	IF NOT(bError) THEN
		ReadBlock(
			NETID 		:= sNetId,
			PORT 		:= nPort,
			IDXGRP 		:= nIDN,
			IDXOFFS 	:= iMIN,
			LEN 		:= cbRead,
			DESTADDR 	:= dwDestAddr_I,
			READ 		:= TRUE,
			TMOUT 		:= tTimeout
		);
		Timeout(IN := FALSE);
	END_IF

10:	(* read min act *)
	ReadBlock(READ := FALSE);

	IF NOT(ReadBlock.BUSY) THEN
		ReadBlock(READ := FALSE);

		IF NOT(ReadBlock.ERR) THEN
			(* done *)
			iState  := 0;
			bBusy   := FALSE;

			ReadBlock(READ := FALSE);
			iRepeats := 0;
		ELSE
			(* Timeout error *)
			IF (ReadBlock.ErrId = 16#745) AND (iRepeats <= 3) THEN
				Timeout(IN := TRUE);

				IF Timeout.Q THEN
					Timeout(IN := FALSE);
					(* retry request 3 times after timeout of 10 ms *)

					ReadBlock(READ := FALSE); (* create rising edge *)
					iRepeats := iRepeats + 1;
					iState	 := 9;
				END_IF

			(* report other errors immeditelly *)
			ELSE
				bError 	:= ReadBlock.ERR;
				nErrId  := ReadBlock.ERRID;
				bBusy   := FALSE;
				iState	:= 0;

				Timeout(IN := FALSE);
				ReadBlock(READ := FALSE);
			END_IF
		END_IF
	END_IF

11:	(* read max init *)
	iState	   	 := 12;
	dwDestAddr_I := dwDestAddr;

	CASE sAttrib.eLength OF
		eLEN_2BYTE:
			cbRead 	 := 2;

		eLEN_4BYTE:
			cbRead	 := 4;

		eLEN_8BYTE:
			cbRead	 := 8;

	ELSE
		bError	 := TRUE;
		nErrId	 := 16#1004; (* Data parameter wrong value size *)
		bBusy	 := FALSE;
		iState 	 := 0;
	END_CASE

	cbRead 	 	:= LIMIT(0, cbRead, cbLen);

	IF NOT(bError) THEN
		ReadBlock(
			NETID 		:= sNetId,
			PORT 		:= nPort,
			IDXGRP 		:= nIDN,
			IDXOFFS 	:= iMAX,
			LEN 		:= cbRead,
			DESTADDR 	:= dwDestAddr_I,
			READ 		:= TRUE,
			TMOUT 		:= tTimeout
		);
		Timeout(IN := FALSE);
	END_IF

12:	(* read max act *)
	ReadBlock(READ := FALSE);

	IF NOT(ReadBlock.BUSY) THEN
		ReadBlock(READ := FALSE);

		IF NOT(ReadBlock.ERR) THEN
			(* done *)
			iState  := 0;
			bBusy   := FALSE;

			ReadBlock(READ := FALSE);
			iRepeats := 0;
		ELSE
			(* Timeout error *)
			IF (ReadBlock.ErrId = 16#745) AND (iRepeats <= 3) THEN
				Timeout(IN := TRUE);

				IF Timeout.Q THEN
					Timeout(IN := FALSE);
					(* retry request 3 times after timeout of 10 ms *)

					ReadBlock(READ := FALSE); (* create rising edge *)
					iRepeats := iRepeats + 1;
					iState	 := 11;
				END_IF

			(* report other errors immeditelly *)
			ELSE
				bError 	:= ReadBlock.ERR;
				nErrId  := ReadBlock.ERRID;
				bBusy   := FALSE;
				iState	:= 0;

				Timeout(IN := FALSE);
				ReadBlock(READ := FALSE);
			END_IF
		END_IF
	END_IF

13: (* Function State *)
	iState 		 := 14;
	dwDestAddr_I := dwDestAddr;
	cbRead		 := cbLen;

	ReadBlock(
		NETID 		:= sNetId,
		PORT 		:= nPort,
		IDXGRP 		:= nIDN,
		IDXOFFS 	:= iFCNSTATE,
		LEN 		:= cbRead,
		DESTADDR 	:= dwDestAddr_I,
		READ 		:= TRUE,
		TMOUT 		:= tTimeout
	);
	Timeout(IN := FALSE);


14:	(* read value act *)
	ReadBlock(READ := FALSE);

	IF NOT(ReadBlock.BUSY) THEN
		ReadBlock(READ := FALSE);

		IF NOT(ReadBlock.ERR) THEN
			(* done *)
			iState	:= 0;
			bBusy	:= FALSE;
			iRepeats 	:= 0;
			ReadBlock(READ := FALSE);
		ELSE
			(* Timeout error *)
			IF (ReadBlock.ErrId = 16#745) AND (iRepeats <= 3) THEN
				Timeout(IN := TRUE);

				IF Timeout.Q THEN
					Timeout(IN := FALSE);
					(* retry request 3 times after timeout of 10 ms *)

					ReadBlock(READ := FALSE); (* create rising edge *)
					iRepeats := iRepeats + 1;
					iState	 := 13;
				END_IF

			(* report other errors immeditelly *)
			ELSE
				bError 	:= ReadBlock.ERR;
				nErrId  := ReadBlock.ERRID;
				bBusy   := FALSE;
				iState	:= 0;

				Timeout(IN := FALSE);
				ReadBlock(READ := FALSE);
			END_IF
		END_IF
	END_IF

ELSE
	(* error *)
	bError	:= TRUE;
	bBusy	:= FALSE;
	iState 	:= 0;
END_CASE

bExecute_I := bExecute;
END_FUNCTION_BLOCK

(* POU IOF_SER_IDN_Write, ST *)
FUNCTION_BLOCK IOF_SER_IDN_Write
VAR_INPUT
	sNetId 				: T_AmsNetId;
	nIDN				: UINT;					(* S: binary 0******* ********, P: binary 1******* ******** *)
	bExecute			: BOOL;					(* starts write with rising edge *)
	nPort				: UINT;					(* sercos axis ads port number *)
	nAttrib				: DWORD;				(* write: 0= Value *)
	cbLen				: UDINT;				(* max lenght of data buffer *)
	dwSrcAddr 			: DWORD;				(* address of data buffer *)
	tTimeout			: TIME := DEFAULT_ADS_TIMEOUT;(* timeout for complete parameter access (e.g. incl. attribute) *)
END_VAR
VAR_OUTPUT
	nAttribRd			: DWORD;
	sAttrib				: ST_SercosParamAttrib;
	bBusy 				: BOOL;
	bError				: BOOL;
	nErrId 				: UDINT;
END_VAR
VAR
	WriteBlock 			: ADSWRITE;
	ReadBlock 			: ADSREAD;
	iState				: INT;
	iRepeats			: INT;
	cbRead				: UDINT;
	cbWrite				: UDINT;
	dwDestAddr			: UDINT;
	nRetVal				: UDINT;
	bExecute_I			: BOOL;
	Timeout				: TON := (PT := T#100ms);
END_VAR
VAR CONSTANT
	iVALUE				: DINT := 0;		(* Parameter Value *)
	iATTRIB				: DINT := 3;		(* Parameter Attribute *)
END_VAR
(* state machine *)
CASE iState OF
0:	(* wait for rising edge *)
	IF bExecute AND NOT(bExecute_I) THEN
		bBusy    	:= TRUE;
		bError 	  	:= FALSE;
		nErrId 	  	:= 0;
		iRepeats 	:= 0;

		Timeout(IN := FALSE);
		ReadBlock(READ := FALSE);
		WriteBlock(WRITE := FALSE);

		IF (nAttrib <> 0) THEN
			sAttrib.nFactor			:= DWORD_TO_UINT(nAttrib          AND 16#0000FFFF); (* bits  0..15 *)
			sAttrib.eLength			:= DWORD_TO_INT(SHR(nAttrib,  16) AND 16#00000007);	(* bits 16..18 *)
			sAttrib.bCommand		:= DWORD_TO_BOOL(SHR(nAttrib, 19) AND 16#00000001);	(* bit  19     *)
			sAttrib.eType			:= DWORD_TO_INT(SHR(nAttrib,  20) AND 16#00000007);	(* bits 20..22 *)
			sAttrib.bReserved1		:= DWORD_TO_BOOL(SHR(nAttrib, 23) AND 16#00000001);	(* bit  23     *)
			sAttrib.nComma			:= DWORD_TO_USINT(SHR(nAttrib,24) AND 16#0000000F); (* bits 24..27 *)
			sAttrib.bWriteProtCP2	:= DWORD_TO_BOOL(SHR(nAttrib, 28) AND 16#00000001);	(* bit  28     *)
			sAttrib.bWriteProtCP3	:= DWORD_TO_BOOL(SHR(nAttrib, 29) AND 16#00000001);	(* bit  29     *)
			sAttrib.bWriteProtCP4	:= DWORD_TO_BOOL(SHR(nAttrib, 30) AND 16#00000001);	(* bit  30     *)
			sAttrib.bReserved2		:= DWORD_TO_BOOL(SHR(nAttrib, 31) AND 16#00000001);	(* bit  31     *)
		END_IF

		IF (nAttrib = 0) OR (sAttrib.eLength = 0) THEN
			(* read attrib first, write afterwards *)
			iState 		:= 1;
			nRetVal 	:= MEMSET(ADR(sAttrib), 0, SIZEOF(sAttrib));
		ELSE
			(* use known attrib, write immediatelly *)
			nAttribRd	:= nAttrib;
			iState 		:= 3;
		END_IF
	END_IF

1:	(* read attrib init *)
	iState 		:= 2;
	nAttribRd	:= 0;
	cbRead 		:= SIZEOF(nAttribRd);
	dwDestAddr 	:= ADR(nAttribRd);

	ReadBlock(
		NETID 		:= sNetId,
		PORT 		:= nPort,
		IDXGRP 		:= nIDN,
		IDXOFFS 	:= iATTRIB,
		LEN 		:= cbRead,
		DESTADDR 	:= dwDestAddr,
		READ 		:= TRUE,
		TMOUT 		:= tTimeout
	);
	Timeout(IN := FALSE);

2:	(* read attrib act *)
	ReadBlock(READ := FALSE);

	IF NOT(ReadBlock.BUSY) THEN
		ReadBlock(READ := FALSE);

		IF NOT(ReadBlock.ERR) THEN
			(* split attribute *)
			sAttrib.nFactor			:= DWORD_TO_UINT(nAttribRd          AND 16#0000FFFF); 	(* bits  0..15 *)
			sAttrib.eLength			:= DWORD_TO_INT(SHR(nAttribRd,  16) AND 16#00000007);	(* bits 16..18 *)
			sAttrib.bCommand		:= DWORD_TO_BOOL(SHR(nAttribRd, 19) AND 16#00000001);	(* bit  19     *)
			sAttrib.eType			:= DWORD_TO_INT(SHR(nAttribRd,  20) AND 16#00000007);	(* bits 20..22 *)
			sAttrib.bReserved1		:= DWORD_TO_BOOL(SHR(nAttribRd, 23) AND 16#00000001);	(* bit  23     *)
			sAttrib.nComma			:= DWORD_TO_USINT(SHR(nAttribRd,24) AND 16#0000000F);	(* bits 24..27 *)
			sAttrib.bWriteProtCP2	:= DWORD_TO_BOOL(SHR(nAttribRd, 28) AND 16#00000001);	(* bit  28     *)
			sAttrib.bWriteProtCP3	:= DWORD_TO_BOOL(SHR(nAttribRd, 29) AND 16#00000001);	(* bit  29     *)
			sAttrib.bWriteProtCP4	:= DWORD_TO_BOOL(SHR(nAttribRd, 30) AND 16#00000001);	(* bit  30     *)
			sAttrib.bReserved2		:= DWORD_TO_BOOL(SHR(nAttribRd, 31) AND 16#00000001);	(* bit  31     *)

			ReadBlock(READ := FALSE);
			iState	 := 3;
			iRepeats := 0;
		ELSE
			(* Timeout error *)
			IF (ReadBlock.ErrId = 16#745) AND (iRepeats <= 3) THEN
				Timeout(IN := TRUE);

				IF Timeout.Q THEN
					Timeout(IN := FALSE);
					(* retry request 3 times after timeout of 10 ms *)

					ReadBlock(READ := FALSE); (* create rising edge *)
					iRepeats := iRepeats + 1;
					iState 	 := 1;
				END_IF

			(* report other errors immeditelly *)
			ELSE
				bError 	:= ReadBlock.ERR;
				nErrId  := ReadBlock.ERRID;
				bBusy   := FALSE;
				iState 	:= 0;

				Timeout(IN := FALSE);
				ReadBlock( READ := FALSE );
			END_IF
		END_IF
	END_IF

3:	(* Write value init *)
	iState := 4;

	CASE sAttrib.eLength OF
		eLEN_2BYTE:
			cbWrite := 2;

		eLEN_4BYTE:
			cbWrite := 4;

		eLEN_8BYTE:
			cbWrite := 8;

		eLEN_V1BYTE, eLEN_V2BYTE, eLEN_V4BYTE, eLEN_V8BYTE:
			(* calculate number of list items *)
			cbWrite	:= 0;
			nRetVal := MEMCPY(ADR(cbWrite), dwSrcAddr, 2);
			cbWrite	:= cbWrite + 4; (* act len & max len *)

	ELSE
		bError	:= TRUE;
		nErrId	:= 16#1004; (* Data parameter wrong value size *)
		bBusy	:= FALSE;
		iState 	:= 0;
	END_CASE

	cbWrite	:= LIMIT(0, cbWrite, cbLen);

	IF NOT(bError) THEN
		WriteBlock(
			NETID 		:= sNetId,
			PORT 		:= nPort,
			IDXGRP 		:= nIDN,
			IDXOFFS 	:= iVALUE,
			LEN 		:= cbWrite,
			SRCADDR 	:= dwSrcAddr,
			WRITE 		:= TRUE,
			TMOUT 		:= tTimeout
		);
		Timeout(IN := FALSE);
	END_IF

4:	(* Write value act *)
	WriteBlock(WRITE := FALSE);

	IF NOT(WriteBlock.BUSY) THEN
		WriteBlock(WRITE := FALSE);

		IF NOT(WriteBlock.ERR) THEN
			(* done *)
			iState := 0;
			bBusy  := FALSE;

			WriteBlock(WRITE := FALSE);
			iRepeats := 0;
		ELSE
			(* Timeout error *)
			IF (WriteBlock.ErrId = 16#745) AND (iRepeats <= 3) THEN
				Timeout(IN := TRUE);

				IF Timeout.Q THEN
					Timeout(IN := FALSE);
					(* retry request 3 times after timeout of 10 ms *)

					WriteBlock(WRITE := FALSE); (* create rising edge *)
					iRepeats := iRepeats + 1;
					iState	 := 3;
				END_IF

			(* report other errors immeditelly *)
			ELSE
				bError 	:= WriteBlock.ERR;
				nErrId  := WriteBlock.ERRID;
				bBusy   := FALSE;
				iState	:= 0;

				Timeout(IN := FALSE);
				WriteBlock(WRITE := FALSE);
			END_IF
		END_IF
	END_IF

ELSE
	(* error *)
	bError	:= TRUE;
	bBusy	:= FALSE;
	iState	:= 0;
END_CASE

bExecute_I := bExecute;
END_FUNCTION_BLOCK

(* POU IOF_SER_DRIVE_BackupEx, ST *)
FUNCTION_BLOCK IOF_SER_DRIVE_BackupEx
VAR_INPUT
	bCheck				: BOOL;
	bBackup				: BOOL;
	bRestore				: BOOL;
	bCRCEnable			: BOOL;
	bStdBackupList		: BOOL 			:= TRUE;
	bUserBackupList		: BOOL;
	sNetId 					: T_AmsNetId;
	nPort					: UINT;
	sComment			: T_MaxString;
	ePath					: E_OpenPath 	:= PATH_BOOTPATH;
	sPathName			: T_MaxString 	:= 'DRIVEPAR.BIN';
	tTimeout				: TIME := DEFAULT_ADS_TIMEOUT;
	bIgnoreParamErr		: BOOL;
END_VAR
VAR_OUTPUT
	bBusy					: BOOL;
	bError					: BOOL;
	nErrId					: UDINT;
	bCheckOK				: BOOL;
	iSkippedParams			: UINT;
	iHandledParams			: UINT;
(*	Function block specific error codes:
	16#1005 = false backup parameter type 
	16#1006 = backup list was not IDN 192 (standard backup) or 0 (userdefined)
*)
END_VAR
VAR_IN_OUT
	arrList					: ST_SercosParamList;
	arrSkippedList			: ST_SercosParamErrList;
END_VAR
VAR CONSTANT
	iVALUE					: DINT := 0;
END_VAR
VAR
	ReadSercosParam			: IOF_SER_IDN_Read;
	WriteSercosParam		: IOF_SER_IDN_Write;

	OpenBackupFile			: FB_FileOpen;
	CloseBackupFile			: FB_FileClose;
	ReadBackupFile			: FB_FileRead;
	WriteBackupFile			: FB_FileWrite;

	eState					: E_SercosBackupState;

	sCheckData				: ST_SercosString;
	wCRC16_CCITT			: WORD;
	wCheckSum				: WORD;

	bCheck_I				: BOOL;
	bBackup_I				: BOOL;
	bRestore_I				: BOOL;
	bCheck_L				: BOOL;
	bBackup_L				: BOOL;
	bRestore_L				: BOOL;
	bUpdateCRC				: BOOL;

	bBackupDone				: BOOL;
	bRestoreDone			: BOOL;

	nListArrIdx				: UINT;
	sListAttrib				: ST_SercosParamAttrib;

	cbLen					: UDINT;
	arrData					: ARRAY [0..65535] OF BYTE;

	nIDN					: UINT;
	nCRCIDN					: UINT := 142;
	bCRCIDNExist			: BOOL;
	bCRCIDNTest				: BOOL := TRUE;
	iIdx					: UINT;

	sParamHeader			: ST_SercosParamHeader;
	cbSize					: UDINT;
	sFileHeader				: ST_SercosFileHeader;
	sParamData				: ST_SercosParamData;

	iActListItem			: UINT;
	iLastListItem			: UINT;
	bEndOfList				: BOOL;

	bFileOpen				: BOOL;
	hFile					: UINT;
	nVersion				: UDINT := 1;
	nRetVal					: UDINT;

	bWrongListType			: BOOL;
	bFileError				: BOOL;
	nFileErrId				: UDINT;
	bIdnError				: BOOL;
	nIdnErrId				: UDINT;
	nIdnAccessId			: UINT;
	iLargeParam				: UINT;
END_VAR
VAR PERSISTENT
	wSavedCRC16_CCITT		: WORD;
	wSavedCheckSum			: WORD;
	sSavedCheckData			: ST_SercosString;
END_VAR
(* state machine *)
CASE eState OF
	eBkup_IDLE:
		bBusy 		 		:= FALSE;

		(* wait for command *)
		IF bCheck AND bCRCIDNTest AND bCRCEnable THEN
			bError			:= FALSE;
			nErrId			:= 0;
			bFileOpen		:= FALSE;
			bFileError		:= FALSE;
			nFileErrId		:= 0;
			bWrongListType	:= FALSE;
			bIdnError		:= FALSE;
			nIdnErrId		:= 0;
			nIdnAccessId	:= 0;
			bEndOfList		:= FALSE;
			eState 			:= eBkup_READ_IDNLIST_INI;
			bBusy			:= TRUE;
			bCheckOK 		:= FALSE;
			iSkippedParams	:= 0;
			iHandledParams	:= 0;
			iLargeParam		:= 0;
			bBackupDone		:= FALSE;
			bRestoreDone	:= FALSE;
			MEMSET(ADR(arrSkippedList), 0, SIZEOF(arrSkippedList));

		ELSIF (bCheck AND NOT(bCheck_I)) AND bCRCEnable AND bCRCIDNExist THEN
			bError			:= FALSE;
			nErrId			:= 0;
			bFileOpen		:= FALSE;
			bFileError		:= FALSE;
			nFileErrId		:= 0;
			bWrongListType	:= FALSE;
			bIdnError		:= FALSE;
			nIdnErrId		:= 0;
			nIdnAccessId	:= 0;
			bEndOfList		:= FALSE;
			eState 			:= eBkup_CHECK_CRC_ACT;
			bBusy			:= TRUE;
			bCheckOK 		:= FALSE;
			bCheck_I 		:= TRUE;
			iSkippedParams	:= 0;
			iHandledParams	:= 0;
			iLargeParam		:= 0;
			bBackupDone		:= FALSE;
			bRestoreDone	:= FALSE;
			MEMSET(ADR(arrSkippedList), 0, SIZEOF(arrSkippedList));

			ReadSercosParam(bExecute := FALSE);
			ReadSercosParam(
				sNetId 		:= sNetId,
				nIDN		:= nCRCIDN,
				bExecute	:= TRUE,
				nMode		:= iVALUE,
				nPort		:= nPort,
				nAttrib		:= 0,
				cbLen		:= SIZEOF(sCheckData),
				dwDestAddr 	:= ADR(sCheckData),
				tTimeout	:= tTimeout
			);
		ELSE
			IF (bBackup AND NOT(bBackup_I)) OR (bRestore AND NOT(bRestore_I)) THEN
				bBackup_L		:= FALSE;
				bRestore_L		:= FALSE;
				bBusy			:= FALSE;
				bError			:= FALSE;
				nErrId			:= 0;
				bFileOpen		:= FALSE;
				bFileError		:= FALSE;
				nFileErrId		:= 0;
				bWrongListType	:= FALSE;
				bIdnError		:= FALSE;
				nIdnErrId		:= 0;
				nIdnAccessId	:= 0;
				bEndOfList		:= FALSE;
				eState 			:= eBkup_READ_IDNLIST_INI;
				bBusy			:= TRUE;
				bUpdateCRC		:= TRUE;
				bCheckOK 		:= FALSE;
				iSkippedParams	:= 0;
				iHandledParams	:= 0;
				iLargeParam		:= 0;
				bBackupDone		:= FALSE;
				bRestoreDone	:= FALSE;
				MEMSET(ADR(arrSkippedList), 0, SIZEOF(arrSkippedList));

				(* initialize CRC16-CCITT and CheckSum *)
				wSavedCRC16_CCITT 			:= 16#FFFF;
				wSavedCheckSum	  			:= 16#0000;
				sSavedCheckData.iActSize	:= 0;
				sSavedCheckData.sString		:= '';

				IF bBackup AND NOT(bBackup_I) THEN
					(* latch backup request *)
					bBackup_L	:= TRUE;
					bRestore_L	:= FALSE;
					bBackup_I 	:= TRUE;

					IF bUserBackupList THEN
						(* calculate number of list items *)
						iLastListItem 	:= arrList.iActCount;
						iLastListItem 	:= iLastListItem / 2;
						iLastListItem 	:= LIMIT(0, iLastListItem, 2047);
						iActListItem	:= 0;
						nListArrIdx		:= 0;
						eState 			:= eBkup_FILEOPEN;

						OpenBackupFile(
							sNetId 		:= sNetId,
							sPathName	:= sPathName,
							nMode		:= FOPEN_MODEWRITE OR FOPEN_MODEBINARY,
							ePath		:= ePath,
							bExecute	:= TRUE,
							tTimeout	:= tTimeout
						);
					END_IF

				ELSIF bRestore AND NOT(bRestore_I) THEN
					(* latch restore request *)
					bBackup_L	:= FALSE;
					bRestore_L	:= TRUE;
					bRestore_I	:= TRUE;

					IF bUserBackupList THEN
						(* calculate number of list items *)
						iLastListItem 	:= arrList.iActCount;
						iLastListItem 	:= iLastListItem / 2;
						iLastListItem 	:= LIMIT(0, iLastListItem, 2047);
						iActListItem	:= 0;
						nListArrIdx		:= 0;
						eState 			:= eBkup_FILEOPEN;

						OpenBackupFile(
							sNetId 		:= sNetId,
							sPathName	:= sPathName,
							nMode		:= FOPEN_MODEREAD OR FOPEN_MODEBINARY,
							ePath		:= ePath,
							bExecute	:= TRUE,
							tTimeout	:= tTimeout
						);
					END_IF
				END_IF
			END_IF
		END_IF

		wCRC16_CCITT 		:= wSavedCRC16_CCITT;
		wCheckSum	 		:= wSavedCheckSum;


	(*** check CRC and CheckSum ***)
	eBkup_CHECK_CRC_ACT:
		ReadSercosParam(bExecute := FALSE);

		IF NOT(ReadSercosParam.bBusy) THEN
			(* not busy anymore *)
			bError	:= ReadSercosParam.bError;
			nErrId	:= ReadSercosParam.nErrId;
			ReadSercosParam(bExecute := FALSE);

			IF bError THEN
				(* error *)
				bIdnError		:= TRUE;
				nIdnErrId		:= nErrId;
				nIdnAccessId	:= nCRCIDN;
				bBusy			:= FALSE;
				eState 			:= eBkup_IDLE;
			ELSE
				(* read done, compare string *)
				bCheckOK 		:= (sCheckData.sString = sSavedCheckData.sString) AND (sCheckData.sString <> '');
				bBusy			:= FALSE;
				eState 			:= eBkup_IDLE;
			END_IF
		END_IF


	(*** read parameter list ***)
	eBkup_READ_IDNLIST_INI:
		(* first scan: initialization with rising edge on bExecute *)
		eState 			:= eBkup_READ_IDNLIST_ACT;

		IF bStdBackupList AND NOT(bCRCIDNTest) THEN
			nIDN		:= 192;
		ELSE
			nIDN		:= 17;
		END_IF

		ReadSercosParam(bExecute := FALSE);
		ReadSercosParam(
			sNetId 		:= sNetId,
			nIDN		:= nIDN,
			bExecute	:= TRUE,
			nMode		:= iVALUE,
			nPort		:= nPort,
			nAttrib		:= 0,
			cbLen		:= SIZEOF(arrList),
			dwDestAddr 	:= ADR(arrList),
			tTimeout	:= tTimeout
		);

	eBkup_READ_IDNLIST_ACT:
		(* following scans: wait for not busy *)
		ReadSercosParam(bExecute := FALSE);

		IF NOT(ReadSercosParam.bBusy) THEN
			(* not busy anymore *)
			bError	:= ReadSercosParam.bError;
			nErrId	:= ReadSercosParam.nErrId;
			ReadSercosParam(bExecute := FALSE);

			IF bError THEN
				(* error *)
				bBackupDone		:= FALSE;
				bRestoreDone	:= FALSE;
				bBackup_L	 	:= FALSE;
				bRestore_L	 	:= FALSE;
				bBusy			:= FALSE;
				eState 			:= eBkup_IDLE;
				bIdnError		:= TRUE;
				nIdnErrId		:= nErrId;
				nIdnAccessId	:= nIDN;
			ELSE
				(* done *)
				sListAttrib		:= ReadSercosParam.sAttrib;

				IF (sListAttrib.eType = eType_ID) AND (sListAttrib.eLength = eLEN_V2BYTE) THEN
					(* calculate number of list items *)
					iLastListItem 	:= arrList.iActCount;
					iLastListItem 	:= iLastListItem / 2;
					iLastListItem 	:= LIMIT(0, iLastListItem, 2047);
					iActListItem	:= 0;
					nListArrIdx		:= 0;

					IF bCRCIDNTest THEN
						bCRCIDNTest  := FALSE;
						bCRCIDNExist := FALSE;

						FOR iIdx := 0 TO iLastListItem DO
							iActListItem := arrList.iList[iIdx];

							IF iActListItem = nCRCIDN THEN
								bCRCIDNExist := TRUE;
								EXIT;
							END_IF
						END_FOR

						IF bBackup_L OR bRestore_L THEN
							eState 	:= eBkup_READ_IDNLIST_INI;
						ELSE
							bBusy	:= FALSE;
							eState 	:= eBkup_IDLE;
						END_IF

					ELSE
						IF bBackup_L THEN
							eState 		:= eBkup_FILEOPEN;

							OpenBackupFile(
								sNetId 		:= sNetId,
								sPathName	:= sPathName,
								nMode		:= FOPEN_MODEWRITE OR FOPEN_MODEBINARY,
								ePath		:= ePath,
								bExecute	:= TRUE,
								tTimeout	:= tTimeout
							);

						ELSIF bRestore_L THEN
							eState 		:= eBkup_FILEOPEN;

							OpenBackupFile(
								sNetId 		:= sNetId,
								sPathName	:= sPathName,
								nMode		:= FOPEN_MODEREAD OR FOPEN_MODEBINARY,
								ePath		:= ePath,
								bExecute	:= TRUE,
								tTimeout	:= tTimeout
							);
						ELSE
							bBusy			:= FALSE;
							eState 			:= eBkup_IDLE;
						END_IF
					END_IF
				ELSE
					bBackupDone		:= FALSE;
					bRestoreDone	:= FALSE;
					bBackup_L	 	:= FALSE;
					bRestore_L	 	:= FALSE;
					bError			:= TRUE;
					nErrId			:= 16#1005;
					bBusy			:= FALSE;
					eState 			:= eBkup_IDLE;
				END_IF
			END_IF
		END_IF


	(*** backup current list ***)
	eBkup_FILEOPEN:
		OpenBackupFile(bExecute	:= FALSE);

		IF NOT(OpenBackupFile.bBusy) THEN
			bError	:= OpenBackupFile.bError;
			nErrId	:= OpenBackupFile.nErrId;
			OpenBackupFile(bExecute	:= FALSE);

			IF bError THEN
				(* error *)
				bBackupDone	:= FALSE;
				bRestoreDone:= FALSE;
				bBackup_L	:= FALSE;
				bRestore_L	:= FALSE;
				nFileErrId	:= nErrId;
				bBusy		:= FALSE;
				eState 		:= eBkup_IDLE;
				bFileOpen	:= FALSE;
				hFile		:= 0;
			ELSE
				bFileOpen	:= TRUE;
				hFile		:= OpenBackupFile.hFile;

				IF bBackup_L THEN
					(* preset header *)
					sFileHeader.nVersion 	 := nVersion;
					IF bUserBackupList THEN
						sFileHeader.nListType 	 := 0;
					ELSE
						sFileHeader.nListType 	 := nIDN;
					END_IF
					sFileHeader.cbCommentLen := SIZEOF(sComment);
					nRetVal 				 := MEMCPY(ADR(sFileHeader.sComment), ADR(sComment), SIZEOF(sComment));

					WriteBackupFile(
						sNetId 		:= sNetId,
						hFile		:= hFile,
						pWriteBuff	:= ADR(sFileHeader),
						cbWriteLen	:= SIZEOF(sFileHeader),
						bExecute	:= TRUE,
						tTimeout	:= tTimeout
					);
					eState 	:= eBkup_BACKUP_WRITE_FILEHEADER;

				ELSIF bRestore_L THEN
					nRetVal := MEMSET(ADR(sFileHeader), 0, SIZEOF(sFileHeader));

					(* load header *)
					ReadBackupFile(
						sNetId 		:= sNetId,
						hFile		:= hFile,
						pReadBuff	:= ADR(sFileHeader),
						cbReadLen	:= SIZEOF(sFileHeader),
						bExecute	:= TRUE,
						tTimeout	:= tTimeout
					);
					eState 	:= eBkup_RESTORE_READ_FILEHEADER;
				END_IF
			END_IF
		END_IF


	(*** backup init ***)
	eBkup_BACKUP_WRITE_FILEHEADER:
		WriteBackupFile(bExecute := FALSE);

		IF NOT(WriteBackupFile.bBusy) THEN
			bError	:= WriteBackupFile.bError;
			nErrId	:= WriteBackupFile.nErrId;
			WriteBackupFile(bExecute := FALSE);

			IF bError THEN
				(* error *)
				bBackupDone	:= FALSE;
				bFileError	:= TRUE;
				nFileErrId	:= nErrId;
				bError		:= FALSE;
				nErrId		:= 0;
				eState 		:= eBkup_FILECLOSE;

				(* backup aborted *)
				CloseBackupFile(
					sNetId 		:= sNetId,
					hFile		:= hFile,
					bExecute	:= TRUE,
					tTimeout	:= tTimeout
				);

			ELSE
				cbSize 	:= WriteBackupFile.cbWrite;
				eState 	:= eBkup_BACKUP_PARAM_INI;
			END_IF
		END_IF

	(* backup current list *)
	eBkup_BACKUP_PARAM_INI:
		IF NOT(bEndOfList) THEN
			(* first scan: initialization with rising edge on bBackup *)
			bBackupDone			:= FALSE;

			(* get parameter *)
			IF (nListArrIdx >= 0) AND (nListArrIdx <= 2047) THEN
				eState 			:= eBkup_BACKUP_PARAM_ACT;
				nIDN 			:= arrList.iList[nListArrIdx];
				nListArrIdx		:= nListArrIdx + 1;

				ReadSercosParam(bExecute := FALSE);
				ReadSercosParam(
					sNetId 		:= sNetId,
					nIDN		:= nIDN,
					bExecute	:= TRUE,
					nMode		:= iVALUE,
					nPort		:= nPort,
					nAttrib		:= 0,
					cbLen		:= SIZEOF(arrData),
					dwDestAddr 	:= ADR(arrData),
					tTimeout	:= tTimeout
				);

			ELSE
				(* wrong index *)
				ReadSercosParam(bExecute := FALSE);
				iActListItem	:= 0;
				bBackupDone		:= FALSE;
				bIdnError		:= TRUE;
				bError			:= FALSE;
				nErrId			:= 0;
				eState 			:= eBkup_FILECLOSE;

				(* backup aborted *)
				CloseBackupFile(
					sNetId 		:= sNetId,
					hFile		:= hFile,
					bExecute	:= TRUE,
					tTimeout	:= tTimeout
				);
			END_IF
		ELSE
			(* backup completed *)
			ReadSercosParam(bExecute := FALSE);
			iActListItem	:= 0;
			eState 			:= eBkup_FILECLOSE;

			CloseBackupFile(
				sNetId 		:= sNetId,
				hFile		:= hFile,
				bExecute	:= TRUE,
				tTimeout	:= tTimeout
			);
		END_IF

	eBkup_BACKUP_PARAM_ACT:
		(* following scans: wait for not busy *)
		ReadSercosParam(bExecute := FALSE);

		IF NOT(ReadSercosParam.bBusy) THEN
			(* not busy anymore *)
			bError				:= ReadSercosParam.bError;
			nErrId				:= ReadSercosParam.nErrId;
			ReadSercosParam(bExecute := FALSE);

			IF bError AND NOT bIgnoreParamErr THEN
				(* error *)
				bBackupDone		:= FALSE;
				bRestoreDone	:= FALSE;
				bIdnError		:= TRUE;
				nIdnErrId		:= nErrId;
				nIdnAccessId	:= nIDN;
				bError			:= FALSE;
				nErrId			:= 0;
				eState 			:= eBkup_FILECLOSE;

				(* backup aborted *)
				CloseBackupFile(
					sNetId 		:= sNetId,
					hFile		:= hFile,
					bExecute	:= TRUE,
					tTimeout	:= tTimeout
				);
			ELSE
				IF NOT bError THEN
					(* save data header *)
					sParamHeader.nIDN	:= ReadSercosParam.nIDN;
					sParamHeader.nAttrib:= ReadSercosParam.nAttribRd;
					sParamHeader.cbSize	:= UDINT_TO_UINT(ReadSercosParam.cbRead);

					IF sParamHeader.cbSize > 4095 THEN
						iLargeParam := iLargeParam + 1;
					END_IF

					(* update CRC16-CCITT and CheckSum *)
					IF nIDN <> nCRCIDN THEN
						wCRC16_CCITT	:= F_CRC16_CCITT(ADR(arrData), sParamHeader.cbSize, wCRC16_CCITT);
						wCheckSum		:= F_CheckSum16(ADR(arrData), sParamHeader.cbSize, wCheckSum);
					END_IF

					WriteBackupFile(
						sNetId 		:= sNetId,
						hFile		:= hFile,
						pWriteBuff	:= ADR(sParamHeader),
						cbWriteLen	:= SIZEOF(sParamHeader),
						bExecute	:= TRUE,
						tTimeout	:= tTimeout
					);

					eState 		:= eBkup_BACKUP_WRITE_HEADER;
				ELSE
					(* ignore param read error *)
					IF iSkippedParams < 2047 THEN
						arrSkippedList.iList[iSkippedParams] := nIDN;
						arrSkippedList.iError[iSkippedParams] := ReadSercosParam.nErrId;
						arrSkippedList.iActCount := arrSkippedList.iActCount + 1;
						arrSkippedList.iMaxCount := arrSkippedList.iActCount;
					END_IF
					iSkippedParams := iSkippedParams + 1;

					(* next item *)
					IF NOT(bEndOfList) THEN
						(* next item *)
						iActListItem		:= iActListItem + 1;
	
						(* backup next parameter *)
						eState 				:= eBkup_BACKUP_PARAM_INI;
	
						IF (iActListItem >= iLastListItem) THEN
							iActListItem	:= 0;
							bEndOfList		:= TRUE;
	
							(* backup completed *)
							ReadSercosParam(bExecute := FALSE);
							CloseBackupFile(
								sNetId 		:= sNetId,
								hFile		:= hFile,
								bExecute	:= TRUE,
								tTimeout	:= tTimeout
							);
							eState 		:= eBkup_FILECLOSE;
						END_IF
					ELSE
						(* backup completed *)
						CloseBackupFile(
							sNetId 		:= sNetId,
							hFile		:= hFile,
							bExecute	:= TRUE,
							tTimeout	:= tTimeout
						);
						ReadSercosParam(bExecute := FALSE);
						eState 		:= eBkup_FILECLOSE;
					END_IF
				END_IF
			END_IF
		END_IF

	eBkup_BACKUP_WRITE_HEADER:
		WriteBackupFile(bExecute := FALSE);

		IF NOT(WriteBackupFile.bBusy) THEN
			bError	:= WriteBackupFile.bError;
			nErrId	:= WriteBackupFile.nErrId;
			WriteBackupFile(bExecute := FALSE);

			IF bError THEN
				(* error *)
				bBackupDone	:= FALSE;
				bFileError	:= TRUE;
				nFileErrId	:= nErrId;
				bError		:= FALSE;
				nErrId		:= 0;
				eState 		:= eBkup_FILECLOSE;

				(* backup aborted *)
				CloseBackupFile(
					sNetId 		:= sNetId,
					hFile		:= hFile,
					bExecute	:= TRUE,
					tTimeout	:= tTimeout
				);
			ELSE
				cbSize := WriteBackupFile.cbWrite;

				(* save data *)
				CASE sParamData.sAttrib.eLength OF
					eLEN_2BYTE,  eLEN_4BYTE,  eLEN_8BYTE,
					eLEN_V1BYTE, eLEN_V2BYTE, eLEN_V4BYTE, eLEN_V8BYTE:
						WriteBackupFile(
							sNetId 		:= sNetId,
							hFile		:= hFile,
							pWriteBuff	:= ADR(arrData),
							cbWriteLen	:= sParamHeader.cbSize,
							bExecute	:= TRUE,
							tTimeout	:= tTimeout
						);
				ELSE
					;
				END_CASE

				eState 		:= eBkup_BACKUP_WRITE_DATA;
			END_IF
		END_IF

	eBkup_BACKUP_WRITE_DATA:
		WriteBackupFile(bExecute := FALSE);

		IF NOT(WriteBackupFile.bBusy) THEN
			bError	:= WriteBackupFile.bError;
			nErrId	:= WriteBackupFile.nErrId;
			WriteBackupFile(bExecute := FALSE);

			IF bError THEN
				(* error *)
				bBackupDone	:= FALSE;
				bFileError	:= TRUE;
				nFileErrId	:= nErrId;
				bError		:= FALSE;
				nErrId		:= 0;
				eState 		:= eBkup_FILECLOSE;

				(* backup aborted *)
				CloseBackupFile(
					sNetId 		:= sNetId,
					hFile		:= hFile,
					bExecute	:= TRUE,
					tTimeout	:= tTimeout
				);
			ELSE
				cbSize 		:= WriteBackupFile.cbWrite;
				iHandledParams	:= iHandledParams + 1;

				(* next item *)
				IF NOT(bEndOfList) THEN
					(* next item *)
					iActListItem		:= iActListItem + 1;

					(* backup next parameter *)
					eState 				:= eBkup_BACKUP_PARAM_INI;

					IF (iActListItem >= iLastListItem) THEN
						iActListItem	:= 0;
						bEndOfList		:= TRUE;

						(* backup completed *)
						ReadSercosParam(bExecute := FALSE);
						CloseBackupFile(
							sNetId 		:= sNetId,
							hFile		:= hFile,
							bExecute	:= TRUE,
							tTimeout	:= tTimeout
						);
						eState 		:= eBkup_FILECLOSE;
					END_IF
				ELSE
					(* backup completed *)
					CloseBackupFile(
						sNetId 		:= sNetId,
						hFile		:= hFile,
						bExecute	:= TRUE,
						tTimeout	:= tTimeout
					);
					ReadSercosParam(bExecute := FALSE);
					eState 		:= eBkup_FILECLOSE;
				END_IF
			END_IF
		END_IF


	(*** restore init ***)
	eBkup_RESTORE_READ_FILEHEADER:
		ReadBackupFile(bExecute := FALSE);

		IF NOT(ReadBackupFile.bBusy) THEN
			bError	:= ReadBackupFile.bError;
			nErrId	:= ReadBackupFile.nErrId;
			ReadBackupFile(bExecute := FALSE);

			IF bError THEN
				(* error *)
				bRestoreDone:= FALSE;
				bFileError	:= TRUE;
				nFileErrId	:= nErrId;
				bError		:= FALSE;
				nErrId		:= 0;
				eState 		:= eBkup_FILECLOSE;

				(* backup aborted *)
				CloseBackupFile(
					sNetId 		:= sNetId,
					hFile		:= hFile,
					bExecute	:= TRUE,
					tTimeout	:= tTimeout
				);
			ELSE
				cbSize 			:= ReadBackupFile.cbRead;
				sComment		:= sFileHeader.sComment;

				IF sFileHeader.nListType = 192 OR sFileHeader.nListType = 0 THEN
					bWrongListType	:= FALSE;

					ReadBackupFile(
						sNetId 		:= sNetId,
						hFile		:= hFile,
						pReadBuff	:= ADR(sParamHeader),
						cbReadLen	:= SIZEOF(sParamHeader),
						bExecute	:= TRUE,
						tTimeout	:= tTimeout
					);
					eState 			:= eBkup_RESTORE_READ_HEADER;
				ELSE
					bWrongListType	:= TRUE;

					(* backup completed *)
					CloseBackupFile(
						sNetId 		:= sNetId,
						hFile		:= hFile,
						bExecute	:= TRUE,
						tTimeout	:= tTimeout
					);
					eState 		:= eBkup_FILECLOSE;
				END_IF
			END_IF
		END_IF

	eBkup_RESTORE_READ_HEADER:
		ReadBackupFile(bExecute := FALSE);

		IF NOT(ReadBackupFile.bBusy) THEN
			bError	:= ReadBackupFile.bError;
			nErrId	:= ReadBackupFile.nErrId;
			ReadBackupFile(bExecute := FALSE);

			IF bError THEN
				(* error *)
				bRestoreDone:= FALSE;
				bFileError	:= TRUE;
				nFileErrId	:= nErrId;
				bError		:= FALSE;
				nErrId		:= 0;
				eState 		:= eBkup_FILECLOSE;

				(* backup aborted *)
				CloseBackupFile(
					sNetId 		:= sNetId,
					hFile		:= hFile,
					bExecute	:= TRUE,
					tTimeout	:= tTimeout
				);
			ELSE
				cbSize := sParamHeader.cbSize;

				IF (ReadBackupFile.cbRead <> 0) THEN
					nRetVal		:= MEMSET(ADR(arrData[0]), 0, SIZEOF(arrData));

					ReadBackupFile(
						sNetId 		:= sNetId,
						hFile		:= hFile,
						pReadBuff	:= ADR(arrData),
						cbReadLen	:= sParamHeader.cbSize,
						bExecute	:= TRUE,
						tTimeout	:= tTimeout
					);
					eState 			:= eBkup_RESTORE_READ_DATA;
				ELSE
					(* backup completed *)
					CloseBackupFile(
						sNetId 		:= sNetId,
						hFile		:= hFile,
						bExecute	:= TRUE,
						tTimeout	:= tTimeout
					);
					bEndOfList	:= TRUE;
					eState 		:= eBkup_FILECLOSE;
				END_IF
			END_IF
		END_IF

	eBkup_RESTORE_READ_DATA:
		ReadBackupFile(bExecute := FALSE);

		IF NOT(ReadBackupFile.bBusy) THEN
			bError		:= ReadBackupFile.bError;
			nErrId		:= ReadBackupFile.nErrId;
			ReadBackupFile(bExecute := FALSE);

			IF bError THEN
				(* error *)
				bRestoreDone:= FALSE;
				bFileError	:= TRUE;
				nFileErrId	:= nErrId;
				bError		:= FALSE;
				nErrId		:= 0;
				eState 		:= eBkup_FILECLOSE;

				(* backup aborted *)
				CloseBackupFile(
					sNetId 		:= sNetId,
					hFile		:= hFile,
					bExecute	:= TRUE,
					tTimeout	:= tTimeout
				);
			ELSE
				IF ReadBackupFile.bEOF THEN
					bEndOfList	:= TRUE;
				END_IF

				cbSize 	:= ReadBackupFile.cbRead;
				eState 	:= eBkup_RESTORE_PARAM_INI;
			END_IF
		END_IF

	(* restore current list item *)
	eBkup_RESTORE_PARAM_INI:
		(* first scan: initialization with rising edge on bBackup *)
		bRestoreDone	:= FALSE;
		eState 			:= eBkup_RESTORE_PARAM_ACT;
		nIDN			:= sParamHeader.nIDN;

		sParamData.nAttrib					:= sParamHeader.nAttrib;

		(* split attribute *)
		sParamData.sAttrib.nFactor			:= DWORD_TO_UINT(sParamHeader.nAttrib AND 16#0000FFFF); 			(* bits  0..15 *)
		sParamData.sAttrib.eLength			:= DWORD_TO_INT(SHR(sParamHeader.nAttrib, 16) AND 16#00000007);		(* bits 16..18 *)
		sParamData.sAttrib.bCommand			:= DWORD_TO_BOOL(SHR(sParamHeader.nAttrib, 19) AND 16#00000001);	(* bit  19     *)
		sParamData.sAttrib.eType			:= DWORD_TO_INT(SHR(sParamHeader.nAttrib, 20) AND 16#00000007);		(* bits 20..22 *)
		sParamData.sAttrib.bReserved1		:= DWORD_TO_BOOL(SHR(sParamHeader.nAttrib, 23) AND 16#00000001);	(* bit  23     *)
		sParamData.sAttrib.nComma			:= DWORD_TO_USINT(SHR(sParamHeader.nAttrib, 24) AND 16#0000000F);	(* bits 24..27 *)
		sParamData.sAttrib.bWriteProtCP2	:= DWORD_TO_BOOL(SHR(sParamHeader.nAttrib, 28) AND 16#00000001);	(* bit  28     *)
		sParamData.sAttrib.bWriteProtCP3	:= DWORD_TO_BOOL(SHR(sParamHeader.nAttrib, 29) AND 16#00000001);	(* bit  29     *)
		sParamData.sAttrib.bWriteProtCP4	:= DWORD_TO_BOOL(SHR(sParamHeader.nAttrib, 30) AND 16#00000001);	(* bit  30     *)
		sParamData.sAttrib.bReserved2		:= DWORD_TO_BOOL(SHR(sParamHeader.nAttrib, 31) AND 16#00000001);	(* bit  31     *)

		CASE sParamData.sAttrib.eLength OF
			eLEN_2BYTE:
				cbLen	:= 2;

			eLEN_4BYTE:
				cbLen	:= 4;

			eLEN_8BYTE:
				cbLen	:= 8;

			eLEN_V1BYTE, eLEN_V2BYTE, eLEN_V4BYTE, eLEN_V8BYTE:
				nRetVal := MEMCPY(ADR(cbLen), ADR(arrData), 2);
				cbLen	:= cbLen + 4; (* act len & max len *)
		ELSE
			cbLen	:= 0;
		END_CASE

		WriteSercosParam(bExecute := FALSE);
		WriteSercosParam(
			sNetId 		:= sNetId,
			nIDN		:= nIDN,
			bExecute	:= TRUE,
			nPort		:= nPort,
			nAttrib		:= sParamData.nAttrib,
			cbLen		:= cbLen,
			dwSrcAddr	:= ADR(arrData),
			tTimeout	:= tTimeout
		);

	eBkup_RESTORE_PARAM_ACT:
		(* following scans: wait for not busy *)
		WriteSercosParam(bExecute := TRUE);

		IF NOT(WriteSercosParam.bBusy) THEN
			(* not busy anymore *)
			bError				:= WriteSercosParam.bError;
			nErrId				:= WriteSercosParam.nErrId;
			WriteSercosParam(bExecute := FALSE);

			IF bError AND NOT bIgnoreParamErr THEN
				(* error *)
				bBackupDone		:= FALSE;
				bRestoreDone	:= FALSE;
				bIdnError		:= TRUE;
				nIdnErrId		:= nErrId;
				nIdnAccessId	:= nIDN;
				bError			:= FALSE;
				nErrId			:= 0;
				eState 			:= eBkup_FILECLOSE;

				(* backup aborted *)
				CloseBackupFile(
					sNetId 		:= sNetId,
					hFile		:= hFile,
					bExecute	:= TRUE,
					tTimeout	:= tTimeout
				);

			ELSE
				IF NOT bError THEN
					iHandledParams	:= iHandledParams + 1;

					IF cbLen > 4095 THEN
						iLargeParam := iLargeParam + 1;
					END_IF

					(* update CRC16-CCITT and CheckSum *)
					IF nIDN <> nCRCIDN THEN
						wCRC16_CCITT	:= F_CRC16_CCITT(ADR(arrData), cbLen, wCRC16_CCITT);
						wCheckSum		:= F_CheckSum16(ADR(arrData), cbLen, wCheckSum);
					END_IF
				ELSE
					(* ignore param write error *)
					IF iSkippedParams < 2047 THEN
						arrSkippedList.iList[iSkippedParams] := nIDN;
						arrSkippedList.iError[iSkippedParams] := WriteSercosParam.nErrId;
						arrSkippedList.iActCount := arrSkippedList.iActCount + 1;
						arrSkippedList.iMaxCount := arrSkippedList.iActCount;
					END_IF
					iSkippedParams := iSkippedParams + 1;
				END_IF

				(* next parameter *)
				iActListItem	:= iActListItem + 1;

				IF NOT(bEndOfList) THEN
					ReadBackupFile(
						sNetId 		:= sNetId,
						hFile		:= hFile,
						pReadBuff	:= ADR(sParamHeader),
						cbReadLen	:= SIZEOF(sParamHeader),
						bExecute	:= TRUE,
						tTimeout	:= tTimeout
					);
					eState 			:= eBkup_RESTORE_READ_HEADER;
				ELSE
					(* backup completed *)
					CloseBackupFile(
						sNetId 		:= sNetId,
						hFile		:= hFile,
						bExecute	:= TRUE,
						tTimeout	:= tTimeout
					);
					WriteSercosParam(bExecute := FALSE);
					eState 		:= eBkup_FILECLOSE;
				END_IF
			END_IF
		END_IF

	(*** done or aborted  ***)
	eBkup_FILECLOSE:
		CloseBackupFile(bExecute := FALSE);

		IF NOT(CloseBackupFile.bBusy) THEN
			bError	:= CloseBackupFile.bError;
			nErrId	:= CloseBackupFile.nErrId;
			CloseBackupFile(bExecute := FALSE);

			IF bError THEN
				(* error *)
				bBackupDone	:= FALSE;
				bRestoreDone:= FALSE;
				bBackup_L	:= FALSE;
				bRestore_L	:= FALSE;
				bBusy		:= FALSE;
				eState 		:= eBkup_IDLE;
			ELSE
				bFileOpen	:= FALSE;
				hFile		:= 0;

				IF bUpdateCRC AND bCRCEnable THEN
					IF NOT(bFileError OR bIdnError) THEN
						sCheckData.sString := 'CRC= ';
						sCheckData.sString := CONCAT(sCheckData.sString, WORD_TO_STRING(wCRC16_CCITT));
						sCheckData.sString := CONCAT(sCheckData.sString, ', ChkSum= ');
						sCheckData.sString := CONCAT(sCheckData.sString, WORD_TO_STRING(wCheckSum));

						IF bBackup_L OR (bRestore_L AND NOT(bWrongListType)) THEN
							ReadSercosParam(bExecute := FALSE);
							ReadSercosParam(
								sNetId 		:= sNetId,
								nIDN		:= nCRCIDN,
								bExecute	:= TRUE,
								nMode		:= iVALUE,
								nPort		:= nPort,
								nAttrib		:= 0,
								cbLen		:= 4,
								dwDestAddr 	:= ADR(sCheckData),
								tTimeout	:= tTimeout
							);

							eState		 := eBkup_UPDT_CRC_INI;
						ELSE
							IF bWrongListType THEN
								bBackupDone := FALSE;
								bRestoreDone:= FALSE;
								bBackup_L	:= FALSE;
								bRestore_L	:= FALSE;
								bError		:= TRUE;
								nErrId		:= 16#1006;	(* backup list was NOT IDN 192 *)
								bBusy		:= FALSE;
								eState 		:= eBkup_IDLE;
							END_IF
						END_IF
					END_IF
				ELSE
					(* done, no CRC and check sum *)
					IF bBackup_L THEN
						bBackup_L	:= FALSE;
						bBackupDone	:= TRUE;
					ELSIF bRestore_L THEN
						bRestore_L	:= FALSE;
						IF NOT bWrongListType THEN
							bRestoreDone:= TRUE;
						ELSE
							bRestoreDone:= FALSE;
						END_IF
					END_IF

					bBusy		:= FALSE;
					eState 		:= eBkup_IDLE;
				END_IF

				IF bFileError THEN
					bError		 := TRUE;
					nErrId		 := nFileErrId;
					bUpdateCRC	 := FALSE;
					bRestoreDone := FALSE;
					bBackupDone	 := FALSE;
					bBackup_L	 := FALSE;
					bRestore_L	 := FALSE;
					bBusy		 := FALSE;
					eState 		 := eBkup_IDLE;
				ELSIF bIdnError THEN
					bError		 := TRUE;
					nErrId		 := nIdnErrId;
					bUpdateCRC	 := FALSE;
					bRestoreDone := FALSE;
					bBackupDone	 := FALSE;
					bBackup_L	 := FALSE;
					bRestore_L	 := FALSE;
					bBusy		 := FALSE;
					eState 		 := eBkup_IDLE;
				END_IF
			END_IF
		END_IF

	eBkup_UPDT_CRC_INI:
		ReadSercosParam(bExecute := FALSE);

		IF NOT(ReadSercosParam.bBusy) THEN
			(* not busy anymore *)
			bError	:= ReadSercosParam.bError;
			nErrId	:= ReadSercosParam.nErrId;
			ReadSercosParam(bExecute := FALSE);

			IF bError THEN
				(* error *)
				bRestoreDone 	:= FALSE;
				bBackupDone	 	:= FALSE;
				bBackup_L	 	:= FALSE;
				bRestore_L	 	:= FALSE;
				bUpdateCRC	 	:= FALSE;
				bIdnError		:= TRUE;
				nIdnErrId		:= nErrId;
				nIdnAccessId	:= nCRCIDN;
				bBusy			:= FALSE;
				eState 			:= eBkup_IDLE;
			ELSE
				sCheckData.iActSize:= LEN(sCheckData.sString);
				sParamData.nAttrib	:= ReadSercosParam.nAttribRd;

				WriteSercosParam(bExecute := FALSE);
				WriteSercosParam(
					sNetId 		:= sNetId,
					nIDN		:= nCRCIDN,
					bExecute	:= TRUE,
					nPort		:= nPort,
					nAttrib		:= sParamData.nAttrib,
					cbLen		:= sCheckData.iActSize + 4,
					dwSrcAddr	:= ADR(sCheckData),
					tTimeout	:= tTimeout
				);

				eState		 := eBkup_UPDT_CRC_ACT;
			END_IF
		END_IF

	eBkup_UPDT_CRC_ACT:
		(* wait for CRC updated *)
		WriteSercosParam(bExecute := FALSE);

		IF NOT(WriteSercosParam.bBusy) THEN
			(* not busy anymore *)
			bError				:= WriteSercosParam.bError;
			nErrId				:= WriteSercosParam.nErrId;
			WriteSercosParam(bExecute := FALSE);
			bUpdateCRC	 		:= FALSE;

			IF bError THEN
				(* error *)
				bRestoreDone 	:= FALSE;
				bBackupDone	 	:= FALSE;
				bBackup_L	 	:= FALSE;
				bRestore_L	 	:= FALSE;
				bBusy			:= FALSE;
				eState 			:= eBkup_IDLE;
				bIdnError		:= TRUE;
				nIdnErrId		:= nErrId;
				nIdnAccessId	:= nIDN;
				bError			:= FALSE;
				nErrId			:= 0;

			ELSE
				(* done *)
				IF bBackup_L THEN
					bBackup_L	:= FALSE;
					bBackupDone	:= TRUE;
				ELSIF bRestore_L THEN
					bRestore_L	:= FALSE;
					bRestoreDone:= TRUE;
				END_IF

				bBusy			:= FALSE;
				eState 			:= eBkup_IDLE;

				(* update CRC16-CCITT and CheckSum *)
				wSavedCRC16_CCITT := wCRC16_CCITT;
				wSavedCheckSum	  := wCheckSum;
				sSavedCheckData	  := sCheckData;
			END_IF
		END_IF

ELSE
	(* undefined state *)
	bRestoreDone:= FALSE;
	bBackupDone	:= FALSE;
	bBackup_L	:= FALSE;
	bRestore_L	:= FALSE;
	bBusy		:= FALSE;
	bError		:= TRUE;
	bUpdateCRC	:= FALSE;
	eState 		:= eBkup_IDLE;
END_CASE

(* clear current data for edge detection *)
bBackup_I 	:= bBackup_I AND bBackup;
bRestore_I 	:= bRestore_I AND bRestore;
bCheck_I 	:= bCheck_I AND bCheck;
END_FUNCTION_BLOCK

(* POU IOF_SER_DRIVE_Reset, ST *)
FUNCTION_BLOCK IOF_SER_DRIVE_Reset
VAR_INPUT
	sNetId 				: T_AmsNetId;(* net id of PC ('' = local PC) *)
	nPort				: UINT;		 (* see System Manager 'IO-Configuration | IO Devices | Sercos Mastert | Sercos Drive | ADS | Port' *)
	bReset			: BOOL;
	tTimeout			: TIME := DEFAULT_ADS_TIMEOUT;
END_VAR
VAR_OUTPUT
	bBusy 				: BOOL;
	bError				: BOOL;
	nErrId 				: UDINT;
END_VAR
VAR
	WriteBlock 		: ADSWRITE;
	iState				: INT;
	iRepeats			: INT;
	nRetVal			: UDINT;
	bReset_I			: BOOL;
	Timeout			: TON := (PT := T#100ms);
	nAttrib				: DWORD;
	iValue				: INT;
END_VAR
(* state machine *)
CASE iState OF
0:	(* wait for rising edge *)
	IF bReset AND NOT(bReset_I) THEN
		bBusy    	:= TRUE;
		bError 	  	:= FALSE;
		nErrId 	  	:= 0;
		iRepeats 	:= 0;
		iState		:= 1;

		Timeout(IN := FALSE);
		WriteBlock(WRITE := FALSE);
	END_IF

1:	(* Write value init *)
	iState 	:= 2;
	iValue	:= 3;

	WriteBlock(
		NETID 		:= sNetId,
		PORT 		:= nPort,
		IDXGRP 		:= 99,		(* = S-0-0099 Drive-Reset-Parameter *)
		IDXOFFS 	:= 8,
		LEN 		:= SIZEOF(iValue),
		SRCADDR 	:= ADR(iValue),
		WRITE 		:= TRUE,
		TMOUT 		:= tTimeout
	);
	Timeout(IN := FALSE);

2:	(* Write value act *)
	WriteBlock(WRITE := FALSE);

	IF NOT(WriteBlock.BUSY) THEN
		WriteBlock(WRITE := FALSE);

		IF NOT(WriteBlock.ERR) THEN
			(* done *)
			iState := 0;
			bBusy  := FALSE;

			WriteBlock(WRITE := FALSE);
			iRepeats := 0;
		ELSE
			(* Timeout error *)
			IF (WriteBlock.ErrId = 16#745) AND (iRepeats <= 3) THEN
				Timeout(IN := TRUE);

				IF Timeout.Q THEN
					Timeout(IN := FALSE);
					(* retry request 3 times after timeout of 10 ms *)

					WriteBlock(WRITE := FALSE); (* create rising edge *)
					iRepeats := iRepeats + 1;
					iState	 := 1;
				END_IF

			(* report other errors immeditelly *)
			ELSE
				bError 	:= WriteBlock.ERR;
				nErrId  := WriteBlock.ERRID;
				bBusy   := FALSE;
				iState	:= 0;

				Timeout(IN := FALSE);
				WriteBlock(WRITE := FALSE);
			END_IF
		END_IF
	END_IF

ELSE
	(* error *)
	bError	:= TRUE;
	bBusy	:= FALSE;
	iState	:= 0;
END_CASE

bReset_I := bReset;
END_FUNCTION_BLOCK

(* POU IOF_SER_GetPhase, ST *)
FUNCTION_BLOCK IOF_SER_GetPhase
VAR_INPUT
	NETID			: T_AmsNetId;
	DEVICEID		: UDINT;
	GET			: BOOL;
	TMOUT		: TIME := DEFAULT_ADS_TIMEOUT;
END_VAR
VAR_OUTPUT
	BUSY			: BOOL;
	ERR			: BOOL;
	ERRID			: UDINT;
	PHASE		: BYTE;
END_VAR
VAR
	ADSREADEX1	: ADSREADEX;
	RisingEdge	: R_TRIG;
	FallingEdge	: F_TRIG;
END_VAR
RisingEdge(CLK:=GET);
IF RisingEdge.Q THEN
	BUSY := TRUE;
	ERR:= FALSE;
	ERRID := 0;
	IF (DEVICEID > 0) AND (DEVICEID <= 255) THEN
		ADSREADEX1(		NETID:=NETID,
						PORT:= AMSPORT_R0_IO,
						IDXGRP:= 16#00005000 + DEVICEID,
						IDXOFFS:= 16#FFFF0100,
						LEN:= SIZEOF(PHASE),
						DESTADDR:= ADR(PHASE),
						READ:=TRUE,
						TMOUT:= TMOUT );
		ADSREADEX1( READ:=FALSE);
	ELSE
		PHASE:=0;
		BUSY := FALSE;
		ERR:=TRUE;
		ERRID :=16#706;(* Parameter value not correct! *)
		RETURN;
	END_IF
ELSE
	ADSREADEX1( READ:=FALSE);
END_IF

FallingEdge( CLK:= ADSREADEX1.BUSY );
IF FallingEdge.Q THEN
	BUSY := FALSE;
	ERR := ADSREADEX1.ERR;
	ERRID := ADSREADEX1.ERRID;

	IF ( ( NOT ERR ) AND ( ADSREADEX1.COUNT_R <> ADSREADEX1.LEN ) ) THEN
		ERR := TRUE;
		ERRID := 16#70B; (* 1803 invalid parameter value(s) *)
	END_IF

	IF ERR THEN
		PHASE:=0;
	END_IF
END_IF
END_FUNCTION_BLOCK

(* POU IOF_SER_ResetErr, ST *)
FUNCTION_BLOCK IOF_SER_ResetErr
VAR_INPUT
	NETID			: T_AmsNetId;
	DEVICEID		: UDINT;
	RESET		: BOOL;
	TMOUT		: TIME := DEFAULT_ADS_TIMEOUT;
END_VAR
VAR_OUTPUT
	BUSY			: BOOL;
	ERR			: BOOL;
	ERRID			: UDINT;
END_VAR
VAR
	ADSWRITE1	: ADSWRITE;
	RisingEdge	: R_TRIG;
	FallingEdge	: F_TRIG;
END_VAR
RisingEdge(CLK:=RESET);
IF RisingEdge.Q THEN
	BUSY := TRUE;
	ERR:= FALSE;
	ERRID:= 0;

	IF DEVICEID > 0 THEN
		ADSWRITE1(		NETID:=NETID,
						PORT:= AMSPORT_R0_IO,
						IDXGRP:= 16#00005000 +DEVICEID,
						IDXOFFS:= 16#FFFF0400,
						LEN:= 0,
						SRCADDR:= 0,
						WRITE:=TRUE,
						TMOUT:= TMOUT );
	ELSE
		BUSY := FALSE;
		ERR:=TRUE;
		ERRID :=16#706;(*Parameter value not correct!*)
		RETURN;
	END_IF
ELSE
	ADSWRITE1( Write:=FALSE);
END_IF

FallingEdge( CLK:= ADSWRITE1.BUSY );
IF FallingEdge.Q THEN
	BUSY := FALSE;
	ERR := ADSWRITE1.ERR;
	ERRID := ADSWRITE1.ERRID;
END_IF
END_FUNCTION_BLOCK

(* POU IOF_SER_SaveFlash, ST *)
FUNCTION_BLOCK IOF_SER_SaveFlash
VAR_INPUT
	NETID			: T_AmsNetId;
	DEVICEID		: UDINT;
	SAVE			: BOOL;
	TMOUT		: TIME := DEFAULT_ADS_TIMEOUT;
END_VAR
VAR_OUTPUT
	BUSY			: BOOL;
	ERR			: BOOL;
	ERRID			: UDINT;
END_VAR
VAR
	ADSWRITE1	: ADSWRITE;
	RisingEdge	: R_TRIG;
	FallingEdge	: F_TRIG;
END_VAR
RisingEdge(CLK:=SAVE);
IF RisingEdge.Q THEN
	BUSY := TRUE;
	ERR := FALSE;
	ERRID := 0;

	IF DEVICEID > 0 THEN
		ADSWRITE1(		NETID:=NETID,
						PORT:= AMSPORT_R0_IO,
						IDXGRP:= 16#00005000 +DEVICEID,
						IDXOFFS:= 16#FFFF0300,
						LEN:= 0,
						SRCADDR:= 0,
						WRITE:=TRUE,
						TMOUT:= TMOUT );
	ELSE
		BUSY := FALSE;
		ERR:=TRUE;
		ERRID :=16#706;(* Parameter value not correct! *)
		RETURN;
	END_IF
ELSE
	ADSWRITE1( Write:=FALSE);
END_IF

FallingEdge( CLK:= ADSWRITE1.BUSY );
IF FallingEdge.Q THEN
	BUSY := FALSE;
	ERR := ADSWRITE1.ERR;
	ERRID := ADSWRITE1.ERRID;
END_IF
END_FUNCTION_BLOCK

(* POU IOF_SER_SetPhase, ST *)
FUNCTION_BLOCK IOF_SER_SetPhase
VAR_INPUT
	NETID			: T_AmsNetId;
	DEVICEID		: UDINT;
	PHASE		: BYTE;
	SET			: BOOL;
	TMOUT		: TIME := DEFAULT_ADS_TIMEOUT;
END_VAR
VAR_OUTPUT
	BUSY			: BOOL;
	ERR			: BOOL;
	ERRID			: UDINT;
END_VAR
VAR
	ADSWRITE1	: ADSWRITE;
	RisingEdge	: R_TRIG;
	FallingEdge	: F_TRIG;
END_VAR
RisingEdge(CLK:=SET);
IF RisingEdge.Q THEN
	BUSY := TRUE;
	ERR := FALSE;
	ERRID := 0;

	IF (PHASE > 4) OR (DEVICEID=0) THEN
		BUSY := FALSE;
		ERR:=TRUE;
		ERRID:=1798; (*invalid parameter value*)
		RETURN;
	ELSE
		ADSWRITE1(		NETID:=NETID,
						PORT:= AMSPORT_R0_IO,
						IDXGRP:= 16#00005000 +DEVICEID,
						IDXOFFS:= 16#FFFF0100,
						LEN:= SIZEOF(PHASE),
						SRCADDR:= ADR(PHASE),
						WRITE:=TRUE,
						TMOUT:= TMOUT);
	END_IF
ELSE
	ADSWRITE1( Write:=FALSE);
END_IF


FallingEdge( CLK:= ADSWRITE1.BUSY );
IF FallingEdge.Q THEN
	BUSY := FALSE;
	ERR := ADSWRITE1.ERR;
	ERRID := ADSWRITE1.ERRID;
END_IF
END_FUNCTION_BLOCK

(* POU SCIT_ActivateConfiguration, ST *)
FUNCTION_BLOCK SCIT_ActivateConfiguration
VAR_INPUT
	NETID 			: T_AmsNetId;
	PORT 			: UINT;
	WRTRD 		: BOOL;
	TMOUT 		: TIME := DEFAULT_ADS_TIMEOUT;
END_VAR
VAR_OUTPUT
	BUSY 			: BOOL;
	ERR 			: BOOL;
	ERRID 			: UDINT;
	RESULT 			: WORD;
	ADDERRORINFO 	: WORD;
END_VAR
VAR
	ADSRDWRT1	: ADSRDWRT;
	BusyFlanke 	: F_TRIG;
	StartFlanke 	: R_TRIG;
	ReadResult 	: ReadResult_t;
	WriteData 		: HLword_t;
END_VAR
	StartFlanke(CLK:=WRTRD );
	IF StartFlanke.Q THEN
		RESULT := 0;
		ADDERRORINFO := 0;
		ReadResult.High1 := 0;
		ReadResult.Low1 := 0;
		ReadResult.High2 := 0;
		ReadResult.Low2 := 0;
		WriteData.High := 0;
		WriteData.Low := 1;
	END_IF

	ADSRDWRT1(	NETID:= NETID,
					PORT:= PORT,
					IDXGRP:= 16#00010001,
					IDXOFFS:= 16#0711,
					WRITELEN:= SIZEOF(WriteData),
					READLEN:= SIZEOF(ReadResult),
					SRCADDR:= ADR(WriteData),
					DESTADDR:= ADR(ReadResult),
					WRTRD:= WRTRD,
					TMOUT:= TMOUT);

	BUSY := ADSRDWRT1.BUSY;
	ERR := ADSRDWRT1.ERR;
	ERRID := ADSRDWRT1.ERRID;

	BusyFlanke(CLK:=BUSY);
	IF BusyFlanke.Q THEN
		RESULT := ReadResult.High1 * 256 + ReadResult.Low1;
		IF RESULT = 0 THEN
			ADDERRORINFO := 0;
		ELSE
			ADDERRORINFO := ReadResult.High2 * 256 + ReadResult.Low2;
		END_IF
	END_IF
END_FUNCTION_BLOCK

(* POU SCIT_AlarmStop, ST *)
FUNCTION_BLOCK SCIT_AlarmStop
VAR_INPUT
	NETID 			: T_AmsNetId;
	PORT 			: UINT;
	WRTRD 		: BOOL;
	TMOUT 		: TIME := DEFAULT_ADS_TIMEOUT;
END_VAR
VAR_OUTPUT
	BUSY 			: BOOL;
	ERR 			: BOOL;
	ERRID 			: UDINT;
	RESULT 			: WORD;
	ADDERRORINFO 	: WORD;
END_VAR
VAR
	ADSRDWRT1		: ADSRDWRT;
	BusyFlanke 		: F_TRIG;
	StartFlanke 	: R_TRIG;
	ReadResult 		: ReadResult_t;
END_VAR
	StartFlanke(CLK:=WRTRD );
	IF StartFlanke.Q THEN
		RESULT := 0;
		ADDERRORINFO := 0;
		ReadResult.High1 := 0;
		ReadResult.Low1 := 0;
		ReadResult.High2 := 0;
		ReadResult.Low2 := 0;
	END_IF

	ADSRDWRT1(	NETID:= NETID,
					PORT:= PORT,
					IDXGRP:= 16#00010001,
					IDXOFFS:= 16#1303,
					WRITELEN:= 0,
					READLEN:= SIZEOF(ReadResult),
					SRCADDR:= 0,
					DESTADDR:= ADR(ReadResult),
					WRTRD:= WRTRD,
					TMOUT:= TMOUT);

	BUSY := ADSRDWRT1.BUSY;
	ERR := ADSRDWRT1.ERR;
	ERRID := ADSRDWRT1.ERRID;

	BusyFlanke(CLK:=BUSY);
	IF BusyFlanke.Q THEN
		RESULT := ReadResult.High1 * 256 + ReadResult.Low1;
		IF RESULT = 0 THEN
			ADDERRORINFO := 0;
		ELSE
			ADDERRORINFO := ReadResult.High2 * 256 + ReadResult.Low2;
		END_IF
	END_IF
END_FUNCTION_BLOCK

(* POU SCIT_ConfDevErrAll, ST *)
FUNCTION_BLOCK SCIT_ConfDevErrAll
VAR_INPUT
	NETID 			: T_AmsNetId;
	PORT 			: UINT;
	WRTRD 		: BOOL;
	TMOUT 		: TIME := DEFAULT_ADS_TIMEOUT;
END_VAR
VAR_OUTPUT
	BUSY 			: BOOL;
	ERR 			: BOOL;
	ERRID 			: UDINT;
	RESULT 			: WORD;
	ADDERRORINFO 	: WORD;
END_VAR
VAR
	ADSRDWRT1		: ADSRDWRT;
	BusyFlanke 		: F_TRIG;
	StartFlanke 	: R_TRIG;

	ReadResult 		: ReadResult_t;
	WriteData 		: DWORD;
END_VAR
	StartFlanke(CLK:=WRTRD );
	IF StartFlanke.Q THEN
		RESULT := 0;
		ADDERRORINFO := 0;
		ReadResult.High1 := 0;
		ReadResult.Low1 := 0;
		ReadResult.High2 := 0;
		ReadResult.Low2 := 0;
		WriteData := 16#00000400;
	END_IF

	ADSRDWRT1(	NETID:= NETID,
					PORT:= PORT,
					IDXGRP:= 16#00010001,
					IDXOFFS:= 16#0714,
					WRITELEN:= SIZEOF(WriteData),
					READLEN:= SIZEOF(ReadResult),
					SRCADDR:= ADR(WriteData),
					DESTADDR:= ADR(ReadResult),
					WRTRD:= WRTRD,
					TMOUT:= TMOUT);

	BUSY := ADSRDWRT1.BUSY;
	ERR := ADSRDWRT1.ERR;
	ERRID := ADSRDWRT1.ERRID;

	BusyFlanke(CLK:=BUSY);
	IF BusyFlanke.Q THEN
		RESULT := ReadResult.High1 * 256 + ReadResult.Low1;
		IF RESULT = 0 THEN
			ADDERRORINFO := 0;
		ELSE
			ADDERRORINFO := ReadResult.High2 * 256 + ReadResult.Low2;
		END_IF
	END_IF
END_FUNCTION_BLOCK

(* POU SCIT_ControlActiveConfiguration, ST *)
FUNCTION_BLOCK SCIT_ControlActiveConfiguration
VAR_INPUT
	NETID 			: T_AmsNetId;
	PORT 			: UINT;
	WRTRD 			: BOOL;
	TMOUT 			: TIME := DEFAULT_ADS_TIMEOUT;
	SWITCH_CODE 	: WORD;
	DEVICE_NO 		: WORD;
END_VAR
VAR_OUTPUT
	BUSY 			: BOOL;
	ERR 			: BOOL;
	ERRID 			: UDINT;
	RESULT 			: WORD;
	ADDERRORINFO 	: WORD;
END_VAR
VAR
	ADSRDWRT1		: ADSRDWRT;
	BusyFlanke 		: F_TRIG;
	StartFlanke 	: R_TRIG;
	ReadResult 		: ReadResult_t;
	WriteData 		: ControlActiveConfiguration_t;
END_VAR
	StartFlanke(CLK:=WRTRD );
	IF StartFlanke.Q THEN
		RESULT := 0;
		ADDERRORINFO := 0;
		ReadResult.High1 := 0;
		ReadResult.Low1 := 0;
		ReadResult.High2 := 0;
		ReadResult.Low2 := 0;
		WriteData.HighSwitchCode := WORD_TO_BYTE(SWITCH_CODE / 256);
		WriteData.LowSwitchCode := WORD_TO_BYTE(SWITCH_CODE);
		WriteData.High1 := 0;
		WriteData.Low1 := 1;
		WriteData.HighDeviceNo := WORD_TO_BYTE(DEVICE_NO / 256);
		WriteData.LowDeviceNo := WORD_TO_BYTE(DEVICE_NO);
	END_IF

	ADSRDWRT1(	NETID:= NETID,
					PORT:= PORT,
					IDXGRP:= 16#00010001,
					IDXOFFS:= 16#0713,
					WRITELEN:= SIZEOF(WriteData),
					READLEN:= SIZEOF(ReadResult),
					SRCADDR:= ADR(WriteData),
					DESTADDR:= ADR(ReadResult),
					WRTRD:= WRTRD,
					TMOUT:= TMOUT);

	BUSY := ADSRDWRT1.BUSY;
	ERR := ADSRDWRT1.ERR;
	ERRID := ADSRDWRT1.ERRID;

	BusyFlanke(CLK:=BUSY);
	IF BusyFlanke.Q THEN
		RESULT := ReadResult.High1 * 256 + ReadResult.Low1;
		IF RESULT = 0 THEN
			ADDERRORINFO := 0;
		ELSE
			ADDERRORINFO := ReadResult.High2 * 256 + ReadResult.Low2;
		END_IF
	END_IF
END_FUNCTION_BLOCK

(* POU SCIT_DeactivateConfiguration, ST *)
FUNCTION_BLOCK SCIT_DeactivateConfiguration
VAR_INPUT
	NETID 			: T_AmsNetId;
	PORT 			: UINT;
	WRTRD 		: BOOL;
	TMOUT 		: TIME := DEFAULT_ADS_TIMEOUT;
END_VAR
VAR_OUTPUT
	BUSY 			: BOOL;
	ERR 			: BOOL;
	ERRID 			: UDINT;
	RESULT 			: WORD;
	ADDERRORINFO 	: WORD;
END_VAR
VAR
	ADSRDWRT1		: ADSRDWRT;
	BusyFlanke 		: F_TRIG;
	StartFlanke 	: R_TRIG;
	ReadResult 		: ReadResult_t;
	WriteData 		: HLword_t;
END_VAR
	StartFlanke(CLK:=WRTRD );
	IF StartFlanke.Q THEN
		RESULT := 0;
		ADDERRORINFO := 0;
		ReadResult.High1 := 0;
		ReadResult.Low1 := 0;
		ReadResult.High2 := 0;
		ReadResult.Low2 := 0;
		WriteData.High := 0;
		WriteData.Low := 1;
	END_IF

	ADSRDWRT1(	NETID:= NETID,
					PORT:= PORT,
					IDXGRP:= 16#00010001,
					IDXOFFS:= 16#0712,
					WRITELEN:= SIZEOF(WriteData),
					READLEN:= SIZEOF(ReadResult),
					SRCADDR:= ADR(WriteData),
					DESTADDR:= ADR(ReadResult),
					WRTRD:= WRTRD,
					TMOUT:= TMOUT);

	BUSY := ADSRDWRT1.BUSY;
	ERR := ADSRDWRT1.ERR;
	ERRID := ADSRDWRT1.ERRID;

	BusyFlanke(CLK:=BUSY);
	IF BusyFlanke.Q THEN
		RESULT := ReadResult.High1 * 256 + ReadResult.Low1;
		IF RESULT = 0 THEN
			ADDERRORINFO := 0;
		ELSE
			ADDERRORINFO := ReadResult.High2 * 256 + ReadResult.Low2;
		END_IF
	END_IF
END_FUNCTION_BLOCK

(* POU SCIT_GetErrorInfo, ST *)
FUNCTION_BLOCK SCIT_GetErrorInfo
VAR_INPUT
	NETID 			: T_AmsNetId;
	PORT 			: UINT;
	WRTRD 		: BOOL;
	TMOUT 		: TIME := DEFAULT_ADS_TIMEOUT;
END_VAR
VAR_OUTPUT
	BUSY 			: BOOL;
	ERR 			: BOOL;
	ERRID 			: UDINT;
	RESULT 			: WORD;
	ERRORCODE 		: WORD;
	ADDERRORINFO 	: WORD;
END_VAR
VAR
	ADSRDWRT1		: ADSRDWRT;
	BusyFlanke 		: F_TRIG;
	StartFlanke 	: R_TRIG;
	WriteData 		: HLword_t;
	ReadResult 		: GetErrorInfo_t;
END_VAR
	StartFlanke(CLK:=WRTRD );
	IF StartFlanke.Q THEN
		RESULT := 0;
		ERRORCODE := 0;
		ADDERRORINFO := 0;
		ReadResult.HighResult := 0;
		ReadResult.LowResult := 0;
		ReadResult.HighEntryCount := 0;
		ReadResult.LowEntryCount := 0;
		ReadResult.HighErrorCode := 0;
		ReadResult.LowErrorCode := 0;
		ReadResult.HighAddErrInfo := 0;
		ReadResult.LowAddErrInfo := 0;

		WriteData.High := 0;
		WriteData.Low := 0;
	END_IF

	ADSRDWRT1(	NETID:= NETID,
					PORT:= PORT,
					IDXGRP:= 16#00010001,
					IDXOFFS:= 16#0316,
					WRITELEN:= 0,
					READLEN:= SIZEOF(ReadResult),
					SRCADDR:= ADR(WriteData),
					DESTADDR:= ADR(ReadResult),
					WRTRD:= WRTRD,
					TMOUT:= TMOUT);

	BUSY := ADSRDWRT1.BUSY;
	ERR := ADSRDWRT1.ERR;
	ERRID := ADSRDWRT1.ERRID;

	BusyFlanke(CLK:=BUSY);
	IF BusyFlanke.Q THEN
		RESULT := ReadResult.HighResult * 256 + ReadResult.LowResult;
		ERRORCODE := ReadResult.HighErrorCode * 256 + ReadResult.LowErrorCode;
		ADDERRORINFO := ReadResult.HighAddErrInfo * 256 + ReadResult.LowAddErrInfo;
	END_IF
END_FUNCTION_BLOCK

(* POU SCIT_StartDataTransfer, ST *)
FUNCTION_BLOCK SCIT_StartDataTransfer
VAR_INPUT
	NETID 			: T_AmsNetId;
	PORT 			: UINT;
	WRTRD 		: BOOL;
	TMOUT 		: TIME := DEFAULT_ADS_TIMEOUT;
END_VAR
VAR_OUTPUT
	BUSY 			: BOOL;
	ERR 			: BOOL;
	ERRID 			: UDINT;
	RESULT 			: WORD;
	ADDERRORINFO 	: WORD;
END_VAR
VAR
	ADSRDWRT1		: ADSRDWRT;
	BusyFlanke 		: F_TRIG;
	StartFlanke 	: R_TRIG;
	ReadResult 		: ReadResult_t;
END_VAR
	StartFlanke(CLK:=WRTRD );
	IF StartFlanke.Q THEN
		RESULT := 0;
		ADDERRORINFO := 0;
		ReadResult.High1 := 0;
		ReadResult.Low1 := 0;
		ReadResult.High2 := 0;
		ReadResult.Low2 := 0;
	END_IF

	ADSRDWRT1(	NETID:= NETID,
					PORT:= PORT,
					IDXGRP:= 16#00010001,
					IDXOFFS:= 16#0701,
					WRITELEN:= 0,
					READLEN:= SIZEOF(ReadResult),
					SRCADDR:= 0,
					DESTADDR:= ADR(ReadResult),
					WRTRD:= WRTRD,
					TMOUT:= TMOUT);

	BUSY := ADSRDWRT1.BUSY;
	ERR := ADSRDWRT1.ERR;
	ERRID := ADSRDWRT1.ERRID;

	BusyFlanke(CLK:=BUSY);
	IF BusyFlanke.Q THEN
		RESULT := ReadResult.High1 * 256 + ReadResult.Low1;
		IF RESULT = 0 THEN
			ADDERRORINFO := 0;
		ELSE
			ADDERRORINFO := ReadResult.High2 * 256 + ReadResult.Low2;
		END_IF
	END_IF
END_FUNCTION_BLOCK

(* POU SCIT_StopDataTransfer, ST *)
FUNCTION_BLOCK SCIT_StopDataTransfer
VAR_INPUT
	NETID 			: T_AmsNetId;
	PORT 			: UINT;
	WRTRD 		: BOOL;
	TMOUT 		: TIME := DEFAULT_ADS_TIMEOUT;
END_VAR
VAR_OUTPUT
	BUSY 			: BOOL;
	ERR 			: BOOL;
	ERRID 			: UDINT;
	RESULT 			: WORD;
	ADDERRORINFO 	: WORD;
END_VAR
VAR
	ADSRDWRT1		: ADSRDWRT;
	BusyFlanke 		: F_TRIG;
	StartFlanke 	: R_TRIG;
	ReadResult 		: ReadResult_t;
	WriteData 		: WORD;
END_VAR
	StartFlanke(CLK:=WRTRD );
	IF StartFlanke.Q THEN
		RESULT := 0;
		ADDERRORINFO := 0;
		ReadResult.High1 := 0;
		ReadResult.Low1 := 0;
		ReadResult.High2 := 0;
		ReadResult.Low2 := 0;
		WriteData := 0;
	END_IF

	ADSRDWRT1(	NETID:= NETID,
					PORT:= PORT,
					IDXGRP:= 16#00010001,
					IDXOFFS:= 16#0702,
					WRITELEN:= SIZEOF(WriteData),
					READLEN:= SIZEOF(ReadResult),
					SRCADDR:= ADR(WriteData),
					DESTADDR:= ADR(ReadResult),
					WRTRD:= WRTRD,
					TMOUT:= TMOUT);

	BUSY := ADSRDWRT1.BUSY;
	ERR := ADSRDWRT1.ERR;
	ERRID := ADSRDWRT1.ERRID;

	BusyFlanke(CLK:=BUSY);
	IF BusyFlanke.Q THEN
		RESULT := ReadResult.High1 * 256 + ReadResult.Low1;
		IF RESULT = 0 THEN
			ADDERRORINFO := 0;
		ELSE
			ADDERRORINFO := ReadResult.High2 * 256 + ReadResult.Low2;
		END_IF
	END_IF
END_FUNCTION_BLOCK
